(* CODESYS project OSKv1.project

Project tree, tasks and I/O mapping:
  Device : SPK1xx[M01], Production association OWEN, order no. 4, version 3.5.11.54
    application Application
      libraries: Standard, * (System); VisuDialogs, * (System); Standard64, * (System); Util, * (System); VisuKeyboard_En-Ru, 1.3.0.0 (PC Prolog); OwenArchiverErrors, 3.5.4.3 (Production association OWEN); Mx110 Assistant, 3.5.4.12 (Production association OWEN)
      task MainTask (cyclic, interval t#20ms, priority 1) calls PLC_PRG, SteamBlow, DryMode, PaintMode, Utils, PID_controller, AnalogSensHandle, Emrg
      task TrendRecordingTask (cyclic, interval 100 ms, priority 31) calls VisuTrendStorageAccess.GlobalInstances.g_TrendRecordingManager.CyclicCall
      task AlarmManagerTask (cyclic, interval 50 ms, priority 31) calls AlarmManager.Alarm_Prg
      task VISU_TASK (cyclic, interval 100 ms, priority 31) calls VisuElems.Visu_Prg
      task OwenArchiver (cyclic, interval T#100ms, priority 10) calls OwenArchiverDrivers.Archive_Prg
      program PLC_PRG [LD]
      visualisation Humidifier
      program PaintMode [ST]
      global variables GVL
      program DryMode [ST]
      Trend Recording Manager
        Trend_Trend1
      visualisation Chiller
      visualisation StartScreen
      visualisation MainMenu
      program SteamBlow [ST]
      visualisation Trend
      visualisation VENT
      visualisation Settings
      Alarm Configuration
        alarm class Error (priority 10, acknowledge REP_ACK)
        alarm class Warning (priority 30, acknowledge REP)
        alarm class Info (priority 100, acknowledge REP)
        AlarmStorage
        text list Emergencies
        alarm group Emergencies
            0 [Error]: Comparison Equal, ExpressionToCompare TRUE, Expression GVL.InNetEmerg - "Авария по защитам"
            1 [Error]: Comparison Equal, ExpressionToCompare TRUE, Expression Emrg.PhaseEmerg - "Аваря по реле контроля фаз"
            2 [Error]: Comparison Equal, ExpressionToCompare TRUE, Expression Emrg.HeatEmerg - "Нет нагрева"
            3 [Error]: Comparison Equal, ExpressionToCompare TRUE, Expression Emrg.PressureEmerg - "Реле давления"
            4 [Error]: Comparison Equal, ExpressionToCompare TRUE, Expression GVL.TempSensError - "Ошибка датчика температуры"
            5 [Error]: Comparison Equal, ExpressionToCompare TRUE, Expression GVL.HumidSensEmerg - "Ошибка датчика влажности"
            6 [Error]: Comparison Equal, ExpressionToCompare TRUE, Expression GVL.PressBoundsEemrg - "Ошибка давления в камере"
      visualisation DryProgs
      program Utils [ST]
      visualisation DeviceCheck
      visualisation DeviceCheck_2
      program PID_controller [ST]
      visualisation Archive
      program Emrg [ST]
      program AnalogSensHandle [ST]
      visualisation Emergencies
      image pool Images
    OwenRTC : OwenRTC, Production association OWEN, version 3.5.11.5001
        input  Application.PLC_PRG.PLC_DATE : ARRAY [0..80] OF BYTE  // Format Date
        input  Application.PLC_PRG.PLC_TIME : ARRAY [0..80] OF BYTE  // Format Time
        unmapped channels: Year, Month, Day, Hour, Minute, Second, Day of Week, Week of Year, UTC Offset, NTP Enabled, NTP Error, System Timer, New Year, New Month, New Day, New Hour, New Minute, New Second, New UTC Offset, Set Settings DT, Enable NTP, Prefer Server
    OwenCloud : OwenCloud, Production association OWEN, version 3.5.11.5001
        unmapped channels: OwenCloud enabled, Enable OwenCloud, Token
    Buzzer : Buzzer, Production association OWEN, version 3.5.11.5001
        unmapped channels: Buzzer enabled, Enable Buzzer
    Drives : Drives, Production association OWEN, version 3.5.11.5001
        input  Application.PLC_PRG.USBMounted : BIT  // MMC Mounted
        input  Application.PLC_PRG.USBUnmountDone : BIT  // MMC Unmount done
        output Application.Utils.DrivesOn : BIT  // Enable Drives
        output Application.PLC_PRG.USBUnmount : BIT  // MMC Unmount
        unmapped channels: FS size, FS used, FS free, USB Mounted, USB Unmount done, USB size, USB used, USB free, MMC size, MMC used, MMC free, USB Unmount
    Network : Network, Production association OWEN, version 3.5.11.5001
        unmapped channels: DHCP enabled, IP, Mask, Gateway, MAC, Hostname, Enable DHCP, New IP, New Mask, New Gateway, New Hostname, Set Settings
    Screen : Screen, Production association OWEN, version 3.5.11.5001
        unmapped channels: Get Brightness, Dim time, Off time, Full brightness, Dim brightness, Off brightness, Dim visu name, Off visu name, On visu name, Wake up
    Debug : Debug, Production association OWEN, version 3.5.11.5001
        unmapped channels: RAM used, RAM free, Open files, Processor usage, Core temp, Enable Debug, Debug pause
    Info : Info, Production association OWEN, version 3.5.11.5002
        unmapped channels: VENDOR, DEVICE, SERIAL, RUNTIME, FIRMWARE, LINUX, TARGET, PROJECT, AUTHOR, VERSION, PROFILE, LASTCHANGES
    Watchdog : Watchdog, Production association OWEN, version 3.5.11.5001
        unmapped channels: Exception Handling, Last Exception Code, Last Exception Description, Last Exception Time, Hardware Watchdog Flag, Reboot
    OwenArchiver : OwenArchiver, Production association OWEN, version 3.5.4.9
        output Application.PLC_PRG.StartArchive : BIT  // Запустить архиватор
        unmapped channels: Команда записи, Запись лога отладки, Путь архивации, Имя архива, Код последней ошибки, Архиватор работает, Использование буфера записи, Размер архива
      CSVFormat : CSVFormat, Production association OWEN, version 3.5.4.9
      REAL_Variable : REAL Variable, Production association OWEN, version 3.5.4.9
          settings: Описание переменной = 'Temperatura v kamere'
          output Application.GVL.ChamberFinalTemp : REAL  // Переменная
      REAL_Variable_1 : REAL Variable, Production association OWEN, version 3.5.4.9
          settings: Описание переменной = 'Vlazhnost'
          output Application.GVL.InAHumInside : REAL  // Переменная
      INT_Variable : INT Variable, Production association OWEN, version 3.5.4.9
          settings: Описание переменной = 'Rezhim raboti'
          output Application.GVL.Mode : INT  // Переменная
      NetEmegAch : BYTE Variable, Production association OWEN, version 3.5.4.9
          settings: Описание переменной = 'Avaria po zachitam'
          output Application.Emrg.NetEmergByte : BYTE  // Переменная
      PhaseEmergArch : BYTE Variable, Production association OWEN, version 3.5.4.9
          settings: Описание переменной = 'Rele cntrolya faz'
          output Application.Emrg.PhaseEmergByte : BYTE  // Переменная
      ChillerEmergArc : BYTE Variable, Production association OWEN, version 3.5.4.9
          settings: Описание переменной = 'Avariya chillera'
          output Application.GVL.InChillerEmerByte : BYTE  // Переменная
      HumidEmergArch : BYTE Variable, Production association OWEN, version 3.5.4.9
          settings: Описание переменной = 'Avariya uvlazhnitelya'
          output Application.GVL.InHumidEmergByte : BYTE  // Переменная
      PressureEmergArch : BYTE Variable, Production association OWEN, version 3.5.4.9
          settings: Описание переменной = 'Rele davleniya'
          output Application.Emrg.PressureEmergByte : BYTE  // Переменная
      UpperFilterArch : BYTE Variable, Production association OWEN, version 3.5.4.9
          settings: Описание переменной = 'Zagrayznenie verhnego filtra'
          output Application.Emrg.UpperFilterOutByte : BYTE  // Переменная
      LowerFilterArch : BYTE Variable, Production association OWEN, version 3.5.4.9
          settings: Описание переменной = 'Zagryaznenie nizhnego filtra'
          output Application.Emrg.LowerFilterOutByte : BYTE  // Переменная
      TempSensErrorArch : BYTE Variable, Production association OWEN, version 3.5.4.9
          settings: Описание переменной = 'Oshibka datchika temperaturi'
          output Application.GVL.TempSensErrorByte : BYTE  // Переменная
      HumidSensEmergArch : BYTE Variable, Production association OWEN, version 3.5.4.9
          settings: Описание переменной = 'Oshibka datchika vlazhnosti'
          output Application.GVL.HumidSensEmergByte : BYTE  // Переменная
      HeatEmergArch : BYTE Variable, Production association OWEN, version 3.5.4.9
          settings: Описание переменной = 'Net nagreva'
          output Application.Emrg.HeatEmergByte : BYTE  // Переменная
      PressureBoundsEmergArch : BYTE Variable, Production association OWEN, version 3.5.4.9
          settings: Описание переменной = 'Davlenie vishlo za ramki'
          output Application.GVL.PressBoundsEemrgByte : BYTE  // Переменная
    Modbus_COM : Modbus COM, 3S - Smart Software Solutions GmbH, version 3.5.11.20
        settings: DataBits = 8; StopBits = 1; ComPort = 1
      Modbus_Master_COM_Port : Modbus Master, COM Port, 3S - Smart Software Solutions GmbH, version 3.5.11.20
          settings: Transmission = 'RTU'; ResponseTimeout = 1000; TimeBetweenFrames = 10; Auto-restart communication = TRUE
        MV110_8A : MV110-8A, Production association OWEN, version 3.5.11.04
            input  Application.GVL.InAChamberTemp : REAL  // Измеренное значение
            input  Application.GVL.InAHExchanger : REAL  // Измеренное значение
            input  Application.GVL.InAEntryTemp : REAL  // Измеренное значение
            input  Application.GVL.InAHumInside : REAL  // Измеренное значение
            input  Application.GVL.InAChambPressure : REAL  // Измеренное значение
            input  Application.GVL.InAHumOutside : REAL  // Измеренное значение
            input  Application.GVL.InAFBHeatGate : REAL  // Измеренное значение
            input  Application.GVL.inAFBCoolGate : REAL  // Измеренное значение
            unmapped channels: Channels1_3State, Channels4_6State, Channels7_8State, Отключить модуль, Флаг ошибки, Код статуса, Код статуса, Код статуса, Код статуса, Код статуса, Код статуса, Код статуса, Код статуса, Циклическое время, Циклическое время, Циклическое время, Циклическое время, Циклическое время, Циклическое время, Циклическое время, Циклическое время
        MU110_16R_K : MU110-16R_K, Production association OWEN, version 3.5.11.04
            settings: SlaveAddress = 17; ResponseTimeout = 1000; UseExtendedFunctionCodes = TRUE
            output Application.GVL.OutInflowFan : BOOL  // Маска выходов (запись).Выход 1
            output Application.GVL.OutExhaustFan : BOOL  // Маска выходов (запись).Выход 2
            output Application.GVL.OutLight1 : BOOL  // Маска выходов (запись).Выход 3
            output Application.GVL.OutLight2 : BOOL  // Маска выходов (запись).Выход 4
            output Application.GVL.OutChiller : BOOL  // Маска выходов (запись).Выход 5
            output Application.GVL.OutHumid : BOOL  // Маска выходов (запись).Выход 6
            output Application.GVL.OutEmergLamp : BOOL  // Маска выходов (запись).Выход 7
            output Application.GVL.OutAirPump : BOOL  // Маска выходов (запись).Выход 8
            output Application.GVL.OutModeGate : BOOL  // Маска выходов (запись).Выход 9
            output Application.GVL.OutHeatGate : BOOL  // Маска выходов (запись).Выход 10
            output Application.GVL.OutCoolGate : BOOL  // Маска выходов (запись).Выход 11
            unmapped channels: rMask, wMask, wAlarmState, wAlarmState, Отключить модуль, Флаг ошибки, Маска выходов (запись), Маска выходов (чтение), Аварийное состояние выходов, Запись аварийного состояния
        MV110_16D_DN : MV110-16D_DN, Production association OWEN, version 3.5.11.04
            settings: SlaveAddress = 18; ResponseTimeout = 1000; UseExtendedFunctionCodes = TRUE
            input  Application.GVL.InChillerPwr : BOOL  // Маска входов.Вход 1
            input  Application.GVL.InChillerPump : BOOL  // Маска входов.Вход 2
            input  Application.GVL.InChillerCompressor : BOOL  // Маска входов.Вход 3
            input  Application.GVL.InChillerEmer : BOOL  // Маска входов.Вход 4
            input  Application.GVL.InHumidPwr : BOOL  // Маска входов.Вход 5
            input  Application.GVL.InHumidEmerg : BOOL  // Маска входов.Вход 6
            input  Application.GVL.InFireSteam : BOOL  // Маска входов.Вход 7
            input  Application.GVL.InModeGatePaint : BOOL  // Маска входов.Вход 9
            input  Application.GVL.InModeGateDry : BOOL  // Маска входов.Вход 10
            input  Application.GVL.InPhaseControl : BOOL  // Маска входов.Вход 11
            input  Application.GVL.InNetEmerg : BOOL  // Маска входов.Вход 12
            input  Application.GVL.InChamberPressure : BOOL  // Маска входов.Вход 13
            input  Application.GVL.InUpperFilter : BOOL  // Маска входов.Вход 14
            input  Application.GVL.InLowerFilter : BOOL  // Маска входов.Вход 15
            unmapped channels: Mask, rCounters, wCounter1, wCounter1, wCounter2, wCounter2, wCounter3, wCounter3, wCounter4, wCounter4, wCounter5, wCounter5, wCounter6, wCounter6, wCounter7, wCounter7, wCounter8, wCounter8, wCounter9, wCounter9, wCounter10, wCounter10, wCounter11, wCounter11, wCounter12, wCounter12, wCounter13, wCounter13, wCounter14, wCounter14, wCounter15, wCounter15, wCounter16, wCounter16, Отключить модуль, Флаг ошибки, Маска входов, Значение счетчика, Запись значения счетчика, Команда на запись,
              Значение счетчика, Запись значения счетчика, Команда на запись, Значение счетчика, Запись значения счетчика, Команда на запись, Значение счетчика, Запись значения счетчика, Команда на запись, Значение счетчика, Запись значения счетчика, Команда на запись, Значение счетчика, Запись значения счетчика, Команда на запись, Значение счетчика, Запись значения счетчика, Команда на запись, Значение счетчика, Запись значения счетчика, Команда на запись, Значение счетчика, Запись значения счетчика, Команда на запись, Значение счетчика, Запись значения счетчика, Команда на запись, Значение счетчика, Запись значения счетчика, Команда на запись, Значение счетчика, Запись значения счетчика, Команда на запись, Значение счетчика, Запись значения счетчика, Команда на запись, Значение счетчика, Запись значения счетчика, Команда на запись, Значение счетчика,
              Запись значения счетчика, Команда на запись, Значение счетчика, Запись значения счетчика, Команда на запись
  text list GlobalTextList
  image pool ImagePool
  5ce3da45-db07-42e7-a21c-a00fff4ed8f6|Gear.png
  5ce3da45-db07-42e7-a21c-a00fff4ed8f6|G:\2019.png
  5ce3da45-db07-42e7-a21c-a00fff4ed8f6|G:\123.png
  5ce3da45-db07-42e7-a21c-a00fff4ed8f6|G:\36185-200.png
  5ce3da45-db07-42e7-a21c-a00fff4ed8f6|123.png
  5ce3da45-db07-42e7-a21c-a00fff4ed8f6|2019.png
  5ce3da45-db07-42e7-a21c-a00fff4ed8f6|36185-200.png
*)

// Device/Application/GVL
{attribute 'qualified_only'}
VAR_GLOBAL
	Mode : INT; // 0 = останов 1 = окраска 2 = сушка 3 = продув по парам 4 = авария
	
	PIDTargetTemp : REAL;
	PIDEnable : BOOL;
	ChamberFinalTemp : REAL;
	HExchangerFinalTemp : REAL;
	EntryFinalTemp : REAL;
	
	HeatBlock : BOOL;
	Emergency : BOOL;
	NotEmerg : bool;
	ExhFanD : INT;
	TempSensError : BOOL;
	TempSensErrorByte : BYTE;
	PressBoundsEemrg : BOOL;
	PressBoundsEemrgByte : BYTE;
	HumidSensEmerg : BOOL;
	HumidSensEmergByte : BYTE;
	
	OutInflowFan : BOOL;
	OutExhaustFan : BOOL;
	OutLight1 : BOOL;
	OutLight2 : BOOL;
	OutChiller : BOOL;
	OutHumid : BOOL;
	OutEmergLamp : BOOL;
	OutModeGate : BOOL;
	OutAirPump : BOOL;
	OutHeatGate : BOOL;
	OutCoolGate : BOOL;
	
	InChillerPwr : BOOL;
	InChillerPump : BOOL;
	InChillerCompressor : BOOL;
	InChillerEmer : BOOL;
	InChillerEmerByte : BYTE;
	
	InHumidPwr : BOOL;
	InHumidEmerg : BOOL;
	InHumidEmergByte : BYTE;
	InFireSteam : BOOL;
	InModeGatePaint : BOOL;
	InModeGateDry : BOOL;
	InPhaseControl : BOOL;
	InNetEmerg : BOOL;
	InChamberPressure : BOOL;
	InUpperFilter : BOOL;
	InLowerFilter : BOOL;
	
	
	InAChamberTemp : REAL;
	InAHExchanger : REAL;
	InAEntryTemp : REAL;
	InAFBHeatGate : REAL;
	inAFBCoolGate : REAL;
	InAHumOutside : REAL;
	InAHumInside : REAL;
	InAChambPressure : REAL;
	
END_VAR

// Device/Application/PLC_PRG
PROGRAM PLC_PRG
VAR
	PLC_DATE : STRING(80);
	PLC_TIME : STRING(80);
	dwLightColorToggle : DWORD := 16#FFFFFF00;
	dwOffColorToggle : DWORD := 16#FFFFFFFF;
	ColorGreen : dword := 16#FF009900;
	xButtonLight1 : BOOL;
	xButtonLight2 : BOOL;
	
	StartArchive : BOOL;
	USBMounted: BOOL;
	USBUnmount : BOOL;
	USBUnmountDone : BOOL;
END_VAR
VAR RETAIN
	Light1Ret: BOOL;
	Light2Ret: BOOL;
END_VAR

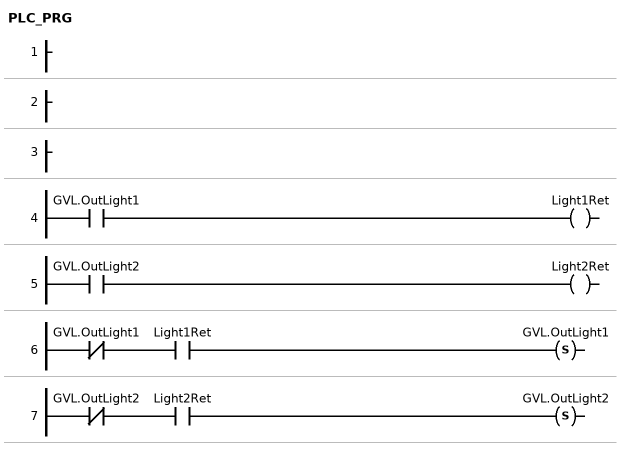
// NETWORK 1

// NETWORK 2

// NETWORK 3

// NETWORK 4
Light1Ret := GVL.OutLight1;

// NETWORK 5
Light2Ret := GVL.OutLight2;

// NETWORK 6
GVL.OutLight1 S= NOT GVL.OutLight1 AND Light1Ret;

// NETWORK 7
GVL.OutLight2 S= NOT GVL.OutLight2 AND Light2Ret;

END_PROGRAM

// Device/Application/SteamBlow
PROGRAM SteamBlow
VAR
	Stage: INT;
	FanCD : TON;
	FanCDStart : BOOL;
	FanCDOut : BOOL;
	
END_VAR

IF .GVL.InFireSteam THEN
	.GVL.Mode := 3;
	Stage := 1;
END_IF

IF (.GVL.InModeGateDry AND Stage = 1) THEN .GVL.OutModeGate := TRUE; END_IF;

IF (.GVL.InModeGatePaint AND Stage = 1) THEN
	.GVL.OutInflowFan := TRUE;
	FanCDStart := TRUE;
	Stage := 2;
END_IF;

FanCD(IN := FanCDStart, PT:= INT_TO_TIME(.GVL.ExhFanD*1000),Q => FanCDOut);

IF FanCDOut THEN
	.GVL.OutExhaustFan := true;
	FanCDStart := FALSE;
END_IF

IF NOT .GVL.InFireSteam AND Stage <> 0 THEN
	.GVL.OutExhaustFan := FALSE;
	.GVL.OutInflowFan := FALSE;
	FanCDStart := FALSE;
	Stage := 0;
	.GVL.Mode := 0;
END_IF

END_PROGRAM

// Device/Application/DryMode
PROGRAM DryMode
VAR
	Modes : ARRAY [0..3] OF WSTRING := ["Пусто","Окраска","Сушка","Продув"];	

	ChosenProg : WORD;
	DryModeM : BOOL;	
	
	NewName : WSTRING;
	SaveName : BOOL;
	ProgChanged : BOOL;	
	SelectedProg: WORD;
	ProgSave : BOOL;
	CurrentName : WSTRING;
	StepTimeLeft : TIME;
	CurStepTime: TIME;
	
	Buffer : ARRAY [1..3,1..10] OF REAL;
	ChooseProg : BOOL;
	
	index: WORD;
	Stage : WORD;
	
	DryTimer : TON;
	DryTimerM : BOOL;
	DryTimerOut : BOOL;
	TempCmp : BOOL;
	
	i: WORD;
	j: WORD;
END_VAR
VAR RETAIN
		// 1 - параметр, 2 - шаг, 3 - программа
	DryPrograms : ARRAY [1..3,1..10,1..10] OF REAL;
	Progs : ARRAY [0..10] OF WSTRING:= ["Выберите программу"];
END_VAR

CurrentName:= Progs[ChosenProg];

IF (ProgChanged = TRUE AND SelectedProg <> 0) THEN
	FOR i:=1 TO 3 BY 1 DO
		FOR j:=1 TO 10 BY 1 DO
			Buffer[i,j] := DryPrograms[i,j,SelectedProg];
		END_FOR;
	END_FOR;
	ProgChanged := FALSE;
END_IF

IF (ProgSave = TRUE AND SelectedProg <> 0) THEN
	FOR i:=1 TO 3 BY 1 DO
		FOR j:=1 TO 10 BY 1 DO
			DryPrograms[i,j,SelectedProg] := Buffer[i,j];
		END_FOR;
	END_FOR;
	ProgSave := FALSE;
END_IF

IF (SaveName = TRUE AND SelectedProg <> 0) THEN
	Progs[SelectedProg] := NewName;
	SaveName := FALSE;
END_IF

IF (ChooseProg = TRUE) THEN
	ChosenProg := SelectedProg;
	ChooseProg := FALSE;
END_IF


IF (Stage = 0 AND .GVL.Mode = 2) THEN index := 1; Stage := 2; DryModeM := TRUE; END_IF; //1

//Если след режим = окр или продув, заслонка = сушка, то выкл вент и заслонку в окраску  2
IF (.GVL.InModeGateDry AND (DryPrograms[1,index,ChosenProg] = 1 OR DryPrograms[1,index,ChosenProg] = 3) AND Stage = 2) THEN 
	.GVL.OutModeGate := TRUE;
	.GVL.OutInflowFan := FALSE;
	.GVL.OutExhaustFan := FALSE;
END_IF;

//Если некст режим = сушка, заслонка = окраска, то выкл вент и заслонку в сушку  3
IF (.GVL.InModeGatePaint AND DryPrograms[1,index,ChosenProg] = 2 AND Stage = 2) THEN 
	.GVL.OutModeGate := FALSE;
	.GVL.OutInflowFan := FALSE;
	.GVL.OutExhaustFan := FALSE;
END_IF;

//Если А[1][index][ChosenProg] = 2 и правильно стоит режимная  4
IF (.GVL.InModeGateDry AND DryPrograms[1,index,ChosenProg] = 2 AND Stage = 2 ) THEN
	IF index > 1 THEN
		IF DryPrograms[2,index,ChosenProg] < DryPrograms[2,index,ChosenProg-1] THEN
			TempCmp := TRUE;
		ELSE TempCmp := FALSE;
		END_IF
	END_IF
	.GVL.PIDTargetTemp := DryPrograms[2,index,ChosenProg];
	.GVL.PIDEnable := TRUE;
	
	.GVL.OutInflowFan := TRUE;
	Stage:=4;
END_IF

// если некст режим = 1 или 3  и правильно стоит режимная  5
IF (.GVL.InModeGatePaint AND (DryPrograms[1,index,ChosenProg] = 1 OR DryPrograms[1,index,ChosenProg] = 3) AND Stage = 2 ) THEN 
	IF index > 1 THEN
		IF DryPrograms[2,index,ChosenProg] < DryPrograms[2,index,ChosenProg-1] THEN
			TempCmp := TRUE;
		ELSE TempCmp := FALSE;
		END_IF
	END_IF
	
	.GVL.OutInflowFan := TRUE;
	.GVL.OutExhaustFan := TRUE;
	DryTimerM := TRUE; //Если режим "вытяжка - вкл", то таймер запускается сразу после начала пункта меню (не дожидаясь достижения температуры).
	Stage := 4;
	.GVL.PIDTargetTemp := DryPrograms[2,index,ChosenProg];
	.GVL.PIDEnable := TRUE;
END_IF;


//если режим - сушка и достигли темп  6
IF (Stage = 4 AND DryPrograms[1,index,ChosenProg] = 2 AND ((.GVL.ChamberFinalTemp < DryPrograms[2,index,ChosenProg] AND TempCmp) OR (.GVL.ChamberFinalTemp > DryPrograms[2,index,ChosenProg] AND NOT TempCmp)) ) THEN
	DryTimerM := TRUE;
END_IF

//В режиме продув остановка по дост темп  7
IF (Stage = 4 AND DryPrograms[1,index,ChosenProg] = 3 AND ((.GVL.ChamberFinalTemp < DryPrograms[2,index,ChosenProg] AND TempCmp) OR (.GVL.ChamberFinalTemp > DryPrograms[2,index,ChosenProg] AND NOT TempCmp))) THEN
	DryTimerM := FALSE;
	Stage := 0;	
	.GVL.OutHeatGate := FALSE;
	.GVL.OutCoolGate := FALSE;
	.GVL.OutInflowFan := FALSE;
	.GVL.OutExhaustFan := FALSE;
	.GVL.Mode := 0;
	DryModeM := FALSE;
	index := 0;
	.GVL.PIDEnable := FALSE;
END_IF

StepTimeLeft := REAL_TO_TIME(DryPrograms[3,index,ChosenProg]*1000) - CurStepTime;

DryTimer(IN := DryTimerM, PT:= REAL_TO_TIME(DryPrograms[3,index,ChosenProg]*1000),ET => CurStepTime,Q => DryTimerOut);

// переход к след шагу по таймеру при режимах 1 и 2   8
IF (DryTimerOut AND DryPrograms[1,index,ChosenProg] <> 3) THEN
	DryTimerM := FALSE;
	Stage := 2;
	index:= index + 1;
END_IF

//если таймер достиг и режим продув то законч работу  9
IF (DryTimerOut AND DryPrograms[1,index,ChosenProg] = 3) THEN
	DryTimerM := FALSE;
	Stage := 0;
	.GVL.OutHeatGate := FALSE;
	.GVL.OutCoolGate := FALSE;
	.GVL.OutInflowFan := FALSE;
	.GVL.OutExhaustFan := FALSE;
	.GVL.Mode := 0;
	DryModeM := FALSE;
	index := 0;
	.GVL.PIDEnable := FALSE;
END_IF

//Handle stop button
IF (.GVL.Mode <> 2 AND stage <> 0) THEN
stage := 0;
.GVL.OutHeatGate := FALSE;
.GVL.OutCoolGate := FALSE;
.GVL.OutExhaustFan := FALSE;
.GVL.OutInflowFan := FALSE;
DryTimerM := FALSE;
DryModeM := FALSE;
index := 0;
.GVL.PIDEnable := FALSE;
END_IF

END_PROGRAM

// Device/Application/PaintMode
PROGRAM PaintMode
VAR
	ExhFanT : TON;
	ExhFanM : BOOL;
	
	ExhFanOut : BOOL;
	
	PaintModeM : BOOL;
	
	ChillT : TON;
	ChillM : BOOL;
	ChillOut : BOOL;
	ChillOK :BOOL;
	ChillHigh : REAL;
	ChillLow : REAL;
	
	Stage : int := 0;
	trig : R_TRIG;

	HumidMax : REAL;
	HumidOk : bool;
	
	TempInc :BOOL;
	TempDec :BOOL;
	TempIncS : BOOL;
	TempDecS : BOOL;
END_VAR
VAR RETAIN
	HumidTarget : INT;
	HumidDiff : INT;
	
	PaintPIDTarget : REAL;
	
	ChillHDiff : REAL;
	ChillLDiff : REAL;
	ChillCD : DINT;
END_VAR

// После нажатия кнопки, проверяется положение режимной заслонки и, при необходимости, она переводится в положение "Окраска".
IF (Stage = 0 AND .GVL.Mode = 1) THEN stage:= 1; PaintModeM := true; END_IF;


IF (.GVL.InModeGateDry AND Stage = 1 AND .GVL.Mode = 1) THEN .GVL.OutModeGate := TRUE; END_IF;

// По окончании перевода, запускается приточный вентилятор и, 
IF (.GVL.InModeGatePaint AND Stage = 1 AND .GVL.HeatBlock = FALSE) THEN 
	Stage := 2;
	.GVL.OutExhaustFan := TRUE;
	ExhFanM:= TRUE;
END_IF;

//через несколько секунд, запускается вытяжной вентилятор и клапан подачи воздуха. 
ExhFanT(IN := ExhFanM, PT:= INT_TO_TIME(.GVL.ExhFanD*1000),Q => ExhFanOut);
IF (ExhFanOut = TRUE AND Stage = 2) THEN 
	.GVL.OutInflowFan := TRUE;
	.GVL.OutAirPump := TRUE;
	Stage := 3;
	ExhFanM:= FALSE;
	.GVL.PIDTargetTemp := PaintPIDTarget;
	.GVL.PIDEnable := TRUE;
END_IF;

//настройка температуры кнопками с панели
IF (TempInc = TRUE)THEN
	PaintPIDTarget := PaintPIDTarget + 1;
	TempInc := FALSE;
END_IF
IF (TempDec = TRUE)THEN
	PaintPIDTarget := PaintPIDTarget - 1;
	TempDec := FALSE;
END_IF
IF (TempIncS = TRUE)THEN
	PaintPIDTarget := PaintPIDTarget + 0.1;
	TempIncS := FALSE;
END_IF
IF (TempDecS = TRUE)THEN
	PaintPIDTarget := PaintPIDTarget - 0.1;
	TempDecS := FALSE;
END_IF

HumidMax := HumidTarget + HumidDiff;

ChillHigh := PaintPIDTarget + ChillHDiff;
ChillLow := PaintPIDTarget + ChillLDiff;

IF (.GVL.InHumidEmerg OR NOT .GVL.InHumidPwr OR .GVL.HumidSensEmerg) THEN
	HumidOk := FALSE;
	.GVL.OutHumid := FALSE;
ELSE HumidOk := TRUE;
END_IF

IF (.GVL.InChillerEmer OR NOT .GVL.InChillerPwr) THEN
	ChillOK := FALSE;
	.GVL.OutChiller := FALSE;
ELSE ChillOK:= TRUE;
END_IF

// В случае, если заслонка находится в положении "0% нагрев", а температура окраски выше заданной более чем на ХХ градуса, включается чиллер
IF (.GVL.InAFBHeatGate < 5 AND stage = 3 AND .GVL.ChamberFinalTemp > ChillHigh AND ChillOK = TRUE) THEN
		.GVL.OutChiller := TRUE;
		Stage := 4;
		.GVL.HeatBlock := TRUE;
END_IF

// И продолжает работать, пока температура не упадет на ХХ градуса ниже температуры ставки. Затем чиллер выключается и запускается внутренний таймер на УУ минут
IF (.GVL.ChamberFinalTemp < ChillLow AND stage = 4) THEN
		.GVL.OutChiller := FALSE;
		ChillM := TRUE;
		stage := 5;
END_IF
ChillT(IN := ChillM, PT:= DINT_TO_TIME(ChillCD*60000),Q => ChillOut);

// По окончании работы этого таймера допускается нагрев воздуха посредством теплообменника
IF (ChillOut = TRUE) THEN
		ChillM := FALSE;
		stage := 0;
		.GVL.HeatBlock := FALSE;
END_IF

// Поддержка влажности
IF (.GVL.InAHumInside > HumidMax AND stage = 3) THEN
		.GVL.OutHumid := FALSE;
END_IF

IF (.GVL.InAHumInside < HumidTarget AND stage = 3 AND HumidOk = TRUE) THEN
		.GVL.OutHumid := TRUE;
END_IF

//Handle stop button
IF (.GVL.Mode <> 1 AND stage <> 0) THEN
stage := 0;
.GVL.OutHeatGate := FALSE;
.GVL.OutCoolGate := FALSE;
.GVL.OutExhaustFan := FALSE;
.GVL.OutInflowFan := FALSE;
.GVL.OutAirPump := FALSE;
.GVL.OutChiller := FALSE;
.GVL.OutHumid := FALSE;
ChillM := FALSE;
ExhFanM := FALSE;
PaintModeM := FALSE;
.GVL.PIDEnable := FALSE;
END_IF

END_PROGRAM

// Device/Application/Utils
PROGRAM Utils
VAR
	GateMode : WSTRING;
	PressureTMR : TON;
	PressureM : BOOL;
	PressureOutM : BOOL;
	
	DrivesOn: BOOL;
	timeR : UINT;
	
	PressureHigh : WORD;
	PressureLow: WORD;
	
	ManualBlock : BOOL;
	
	ColorYelllow : DWORD := 16#FFFFFF00;
	ColorWhite : DWORD := 16#FFFFFFFF;
	ColorGreen : DWORD := 16#FF009900;
	ColorRed : DWORD := 16#FFFF3300;
	
	CurrentChillerColor : DWORD;
	CurrentHumidColor: DWORD;
	CurrentVentColor: DWORD;
	
	ModeGateImg : BOOL;
	NotInflowFan : BOOL;
	NotExhaustFan : BOOL;
END_VAR

IF .GVL.InModeGateDry THEN
	ModeGateImg := FALSE;
ELSIF .GVL.InModeGatePaint THEN
	ModeGateImg := TRUE;
END_IF;

DrivesOn:=true;

NotInflowFan := NOT .GVL.OutInflowFan;
NotExhaustFan := NOT .GVL.OutExhaustFan;

IF .GVL.InChillerEmer THEN
	CurrentChillerColor := ColorRed;
ELSIF .GVL.OutChiller THEN
	CurrentChillerColor := ColorGreen;
ELSE
	CurrentChillerColor := ColorWhite;
END_IF;

IF .GVL.InHumidEmerg THEN
	CurrentHumidColor := ColorRed;
ELSIF .GVL.OutHumid THEN
	CurrentHumidColor := ColorGreen;
ELSE
	CurrentHumidColor := ColorWhite;
END_IF;

IF .GVL.Mode > 2 THEN
	CurrentVentColor := ColorRed;
ELSIF .GVL.Mode > 0 THEN
	CurrentVentColor := ColorGreen;
ELSE
	CurrentVentColor := ColorWhite;
END_IF;

IF .GVL.InModeGateDry THEN
GateMode := "Сушка";
ELSIF .GVL.InModeGatePaint THEN
        GateMode := "Окраска";
ELSE
        GateMode := "Переход";
END_IF;


IF (.GVL.OutInflowFan OR .GVL.OutExhaustFan) AND (.GVL.InAChambPressure > PressureHigh OR .GVL.InAChambPressure < PressureLow) THEN
	PressureM := TRUE;
ELSE
	PressureM := FALSE;
END_IF;

PressureTMR(IN := PressureM, PT:= INT_TO_TIME(20000),Q => PressureOutM);

IF PressureOutM THEN
	.GVL.PressBoundsEemrg := TRUE;
ELSE .GVL.PressBoundsEemrg := FALSE;
END_IF

IF .GVL.Mode <> 0 THEN
	ManualBlock := TRUE;
ELSE ManualBlock := FALSE;
END_IF

END_PROGRAM

// Device/Application/PID_controller
PROGRAM PID_controller
VAR
	PeriodicTMR : TON;
	TMRIn : BOOL;
	TMROut : BOOL;
	TMRCurr : TIME;

	Delta : REAL;
	PIDArray : ARRAY [1..11] OF REAL;
	ArraySum : REAL;
	
	PropComponent : REAL;
	IntComponent : REAL;
	FinalEqus : REAL;
	FinalResult : REAL;
	
	i : INT;
END_VAR
VAR RETAIN
	KI : WORD;
	KP : WORD;
	Tau : WORD;
END_VAR

PeriodicTMR(IN := TMRIn, PT:= WORD_TO_TIME(Tau*1000),ET => TMRCurr,Q => TMROut);
IF TMRIn =  FALSE AND .GVL.PIDEnable = TRUE THEN
	TMRIn := TRUE;
END_IF
IF .GVL.PIDEnable = FALSE THEN
	FOR i:=1 TO 10 BY 1 DO
		PIDArray[i] := 0;
	END_FOR;
END_IF
IF TMROut THEN
	ArraySum := 0;
	Delta := .GVL.ChamberFinalTemp - .GVL.PIDTargetTemp;
	PIDArray[11] := Delta;
	FOR i:=1 TO 10 BY 1 DO
		PIDArray[i] := PIDArray[i+1];
		ArraySum:=ArraySum+PIDArray[i];
	END_FOR;
	
	PropComponent := Delta * KP;
	IntComponent := ArraySum * KI;
	
	FinalEqus := (PropComponent + IntComponent) / 100;
	
	IF FinalEqus > 100 THEN
		FinalResult := 100;
	ELSIF FinalEqus < -100 THEN
		FinalResult := -100;
		ELSE FinalResult := FinalEqus;
	END_IF
	TMRIn := FALSE;
END_IF

IF .GVL.PIDEnable THEN
	IF FinalResult < 0 THEN
		IF .GVL.inAFBHeatGate <> FinalResult THEN
			.GVL.OutHeatGate := TRUE;
		ELSE .GVL.OutHeatGate := FALSE;
		END_IF
	ELSIF .GVL.inAFBCoolGate <> FinalResult THEN
		.GVL.OutCoolGate := TRUE;
		.GVL.OutHeatGate := TRUE;
		ELSE .GVL.OutCoolGate := FALSE;
			.GVL.OutHeatGate := FALSE;
	END_IF
END_IF

END_PROGRAM

// Device/Application/AnalogSensHandle
PROGRAM AnalogSensHandle
VAR
END_VAR

IF .GVL.TempSensError THEN
	.GVL.ChamberFinalTemp := .GVL.InAEntryTemp / 10;
ELSE .GVL.ChamberFinalTemp := .GVL.InAChamberTemp / 10;
END_IF

GVL.EntryFinalTemp := .GVL.InAEntryTemp /10;
GVL.HExchangerFinalTemp := GVL.InAHExchanger /10;

END_PROGRAM

// Device/Application/Emrg
PROGRAM Emrg
VAR
	PressureEmerg : BOOL; // авария по давлению 4
	PressureEmergByte : BYTE;
	NetEmerg : BOOL ; // авария по реле контроля фаз 1 
	NetEmergByte : BYTE;
	HeatEmerg : BOOL; 
	HeatEmergByte : BYTE;
	PhaseEmerg : BOOL;
	PhaseEmergByte : BYTE;
	                    
	
	PressEmergInv : BOOL;
	PressEmergTON : TON;
	PressEmergStart: BOOL;
	PressEmergOut : BOOL;
	
	PressRelEmergInv : BOOL;
	PressRelEmergTON : TON;
	PressRelEmergStart: BOOL;
	PressRelEmergOut : BOOL;
	
	UpperFilter : TON;
	UpperFilterStart: BOOL;
	UpperFilterOut : BOOL;
	UpperFilterOutByte : BYTE;
	
	LowerFilter : TON;
	LowerFilterStart: BOOL;
	LowerFilterOut : BOOL;
	LowerFilterOutByte : BYTE;
	
	UpperFilterInv : BOOL;
	LowerFilterInv : BOOL;
	
	AcknSelected : BOOL;
	AcknVisible : BOOL;
	EmergHistory : BOOL;
	EmergFixedPos : BOOL;
	
	
END_VAR

PressEmergInv := NOT .GVL.InChamberPressure;
UpperFilterInv := NOT .GVL.InUpperFilter;
LowerFilterInv := NOT .GVL.InLowerFilter;
.GVL.NotEmerg := NOT .GVL.Emergency;

PressureEmergByte := BOOL_TO_BYTE(PressureEmerg);
NetEmergByte:= BOOL_TO_BYTE(NetEmerg);
HeatEmergByte:= BOOL_TO_BYTE(HeatEmerg);
PhaseEmergByte:= BOOL_TO_BYTE(PhaseEmerg);
UpperFilterOutByte := BOOL_TO_BYTE(UpperFilterOut);
LowerFilterOutByte := BOOL_TO_BYTE(LowerFilterOut);
.GVL.TempSensErrorByte := BOOL_TO_BYTE(.GVL.TempSensError);
.GVL.PressBoundsEemrgByte := BOOL_TO_BYTE(.GVL.PressBoundsEemrg);
.GVL.HumidSensEmergByte := BOOL_TO_BYTE(.GVL.HumidSensEmerg);
.GVL.InChillerEmerByte := BOOL_TO_BYTE(.GVL.InChillerEmer);
.GVL.InHumidEmergByte := BOOL_TO_BYTE(.GVL.InHumidEmerg);

//Светофор
.GVL.OutEmergLamp := .GVL.Emergency;
//Общий стоп и запрет
IF .GVL.Emergency THEN
	.GVL.Mode := 4;
END_IF

// Авария по защитам, останов
IF .GVL.InNetEmerg THEN
	NetEmerg := TRUE;
	.GVL.Emergency := TRUE;
ELSE NetEmerg := FALSE;
END_IF

IF .GVL.InPhaseControl THEN
	PhaseEmerg := TRUE;
	.GVL.Emergency := TRUE;
ELSE PhaseEmerg := FALSE;
END_IF

//Авария датчика температуры
IF .GVL.InAChamberTemp > 2000 OR .GVL.InAChamberTemp < -500 THEN
	.GVL.TempSensError := TRUE;
ELSE .GVL.TempSensError := FALSE;
END_IF

//Авария датчика влажности
IF .GVL.InAHumInside > 1000 OR .GVL.InAHumInside < 0 THEN
	.GVL.HumidSensEmerg := TRUE;
	.GVL.Emergency := TRUE;
ELSE .GVL.HumidSensEmerg := FALSE;
END_IF

//Нет нагрева
IF .GVL.InAHExchanger < 200 THEN
	HeatEmerg := TRUE;
	.GVL.Emergency := TRUE;
ELSE HeatEmerg := FALSE;
END_IF

// Задержка срабатывания аварии давления
PressEmergTON(IN := PressEmergStart, PT := INT_TO_TIME(10000), Q=> PressEmergOut);
IF .GVL.OutInflowFan OR .GVL.OutExhaustFan THEN
	PressEmergStart := TRUE;
END_IF
IF PressEmergOut THEN
	PressEmergStart := FALSE;
END_IF

// Авария давления, останов
IF NOT PressEmergStart AND PressEmergInv THEN
	PressureEmerg := TRUE;;
	.GVL.Emergency := TRUE;
ELSE PressureEmerg := FALSE;
END_IF

//Грязный фильтр, индикация 
IF LowerFilterInv THEN
	LowerFilterStart := TRUE;
ELSE LowerFilterStart := FALSE;
END_IF
// грязынй фильтр индикация
IF UpperFilterInv THEN
	UpperFilterStart := TRUE;
ELSE UpperFilterStart := FALSE;
END_IF
LowerFilter(IN := LowerFilterStart, PT := INT_TO_TIME(10000), Q=> LowerFilterOut); // авария грязный фильтр 6
UpperFilter(IN := UpperFilterStart, PT := INT_TO_TIME(10000), Q=> UpperFilterOut); // авария грязный фильтр 5

//сброс глобальной ошибки при отсутствии ош
IF NOT PressureEmerg AND NOT NetEmerg AND NOT PhaseEmerg AND NOT .GVL.InNetEmerg AND NOT .GVL.TempSensError AND NOT .GVL.HumidSensEmerg AND NOT .GVL.PressBoundsEemrg AND NOT HeatEmerg AND .GVL.Mode=4 THEN
	.GVL.Emergency := FALSE;
	.GVL.Mode := 0;
END_IF

END_PROGRAM

// Device/Application/Humidifier
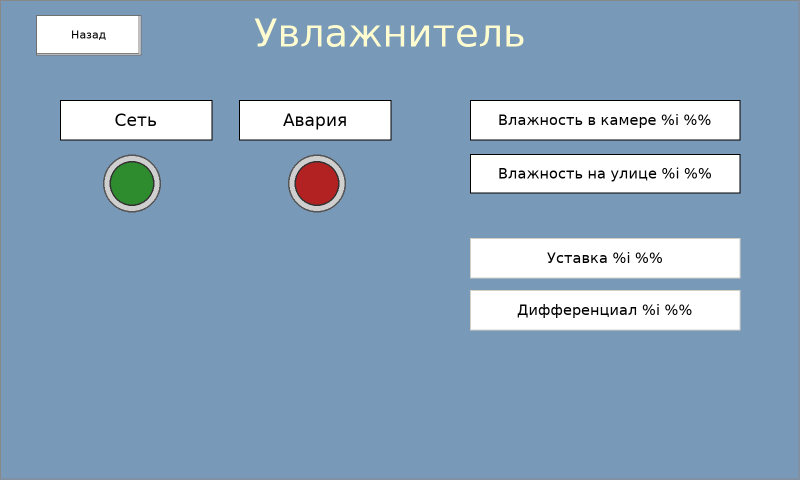
VISUALIZATION Humidifier  // 800x480
    Button (36,15 105x40), "Назад"
        OnMouseClick:  Assign=StartScreen, Type=Assignment
    Label (157,10 466x46), "Увлажнитель"
    Lamp1 (98,150 68x67), variable: GVL.InHumidPwr, style: Lamp-Lamp1-Green
    Lamp1 (283,150 68x67), variable: GVL.InHumidEmerg, style: Lamp-Lamp1-Red
    Rectangle (60,100 152x40), "Сеть"
    Rectangle (239,100 152x40), "Авария"
    Rectangle (470,100 270x40), "Влажность в камере %i %%", text variable: GVL.InAHumInside
    Rectangle (470,154 270x39), "Влажность на улице %i %%", text variable: GVL.InAHumOutside
    Textfield (470,238 270x40), "Уставка %i %%", text variable: PaintMode.HumidTarget
        OnMouseClick: write the text variable via Default, min 0, max 100
    Textfield (470,290 270x40), "Дифференциал %i %%", text variable: PaintMode.HumidDiff
        OnMouseClick: write the text variable via Default, min 0, max 100
END_VISUALIZATION

// Device/Application/Chiller
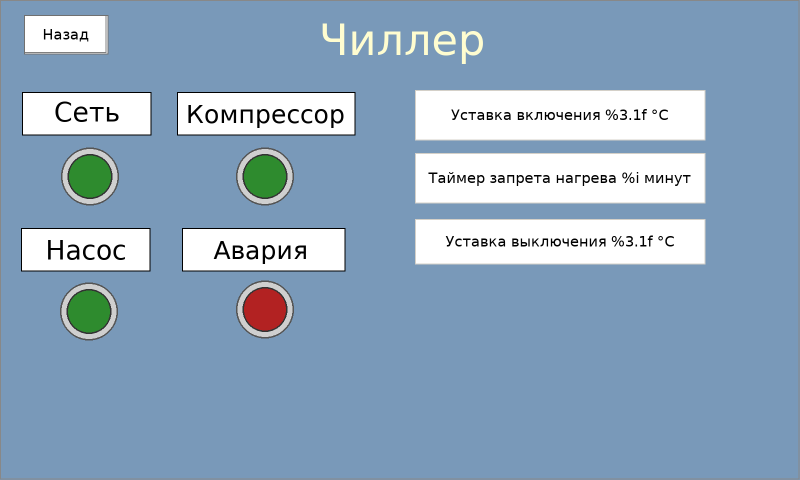
VISUALIZATION Chiller  // 800x480
    Lamp1 (56,143 68x67), variable: GVL.InChillerPwr, style: Lamp-Lamp1-Green
    Rectangle (22,92 129x43)
    Label (29,95 116x34), "Сеть"
    Lamp1 (55,278 68x67), variable: GVL.InChillerPump, style: Lamp-Lamp1-Green
    Rectangle (21,228 129x43)
    Label (28,233 116x34), "Насос"
    Lamp1 (231,143 68x67), variable: GVL.InChillerCompressor, style: Lamp-Lamp1-Green
    Rectangle (177,92 178x43)
    Label (181,97 169x34), "Компрессор"
    Lamp1 (231,276 68x67), variable: GVL.InChillerEmer, style: Lamp-Lamp1-Red
    Rectangle (182,228 163x43)
    Label (196,233 130x34), "Авария"
    Button (24,15 84x39), "Назад"
        OnMouseClick:  Assign=StartScreen, Type=Assignment
    Label (294,14 217x52), "Чиллер"
    Textfield (415,90 290x50), "Уставка включения %3.1f °C", text variable: PaintMode.ChillHDiff
        OnMouseClick: write the text variable via Default, min -50, max 150
    Textfield (415,219 290x45), "Уставка выключения %3.1f °C", text variable: PaintMode.ChillLDiff
        OnMouseClick: write the text variable via Default, min -50, max 150
    Textfield (415,153 290x50), "Таймер запрета нагрева %i минут", text variable: PaintMode.ChillCD
        OnMouseClick: write the text variable via Default, min -50, max 150
END_VISUALIZATION

// Device/Application/StartScreen
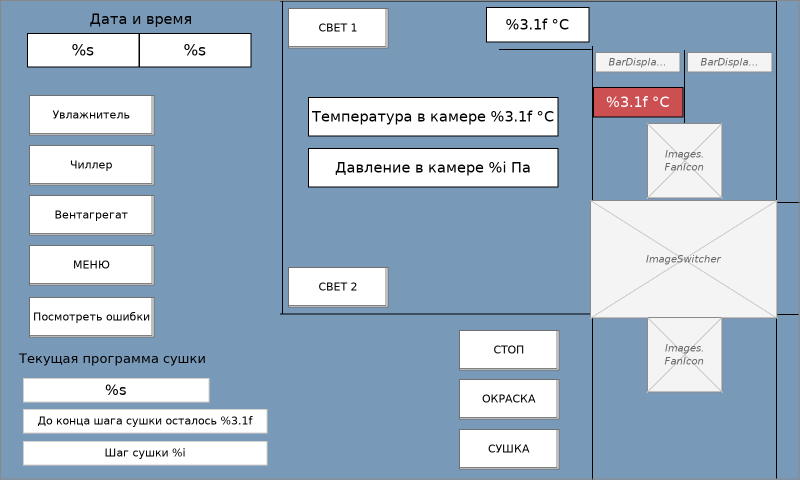
VISUALIZATION StartScreen  // 800x480
    Rectangle (593,87 90x30), "%3.1f °С", text variable: GVL.HExchangerFinalTemp
    Button (459,330 100x40), "СТОП"
        OnMouseClick: execute { .GVL.Mode := 0; }
    Button (459,379 100x40), "ОКРАСКА", colour toggle: PaintMode.PaintModeM
        p2175578022: PLC_PRG.dwOffColorToggle
        p573394764: PLC_PRG.ColorGreen
        OnMouseClick: execute {
            IF (.GVL.Mode = 0) THEN
            .GVL.Mode := 1;
            END_IF;
        }
    Button (459,429 100x40), "СУШКА", colour toggle: DryMode.DryModeM
        p2175578022: PLC_PRG.dwOffColorToggle
        p573394764: PLC_PRG.ColorGreen
        OnMouseClick: execute {
            IF (.GVL.Mode = 0) THEN
            	.GVL.Mode :=2;
            END_IF
        }
    Button (288,8 100x40), "СВЕТ 1", colour toggle: GVL.OutLight1
        p573394764: PLC_PRG.dwLightColorToggle
        p2175578022: PLC_PRG.dwOffColorToggle
        toggle GVL.OutLight1
    Button (288,267 100x40), "СВЕТ 2", colour toggle: GVL.OutLight2
        p573394764: PLC_PRG.dwLightColorToggle
        p2175578022: PLC_PRG.dwOffColorToggle
        toggle GVL.OutLight2
    Button (29,95 125x40), "Увлажнитель"
        p2175578022: Utils.CurrentHumidColor
        OnMouseClick:  Assign=Humidifier, Type=Assignment
    Button (29,145 125x40), "Чиллер"
        p2175578022: Utils.CurrentChillerColor
        OnMouseClick:  Assign=Chiller, Type=Assignment
    Button (29,195 125x40), "Вентагрегат"
        p2175578022: Utils.CurrentVentColor
        OnMouseClick:  Assign=VENT, Type=Assignment
    Button (29,245 125x40), "МЕНЮ"
        OnMouseClick:  Assign=MainMenu, Type=Assignment
    Rectangle (308,97 250x39), "Температура в камере %3.1f °C", text variable: GVL.ChamberFinalTemp
    Rectangle (308,148 250x39), "Давление в камере %i Па", text variable: GVL.InAChambPressure
    Rectangle (139,33 112x34), "%s", text variable: PLC_PRG.PLC_TIME
    Rectangle (27,33 112x34), "%s", text variable: PLC_PRG.PLC_DATE
    Label (43,1 196x36), "Дата и время"
    Label (23,346 179x25), "Текущая программа сушки"
    Textfield (23,378 186x24), "%s", text variable: DryMode.CurrentName
    Textfield (23,409 244x24), "До конца шага сушки осталось %3.1f", text variable: DryMode.StepTimeLeft
    Button (29,297 125x40), "Посмотреть ошибки"
        OnMouseClick:  Assign=Emergencies, Type=Assignment
    Textfield (23,441 244x24), "Шаг сушки %i", text variable: DryMode.index
    Line (800,431)
    Line (774,314) (799,314)
    Line (776,314) (776,479)
    Line (592,314) (592,480)
    Line (774,202) (800,202)
    Line (592,314) (280,314)
    Line (776,1) (280,1)
    Line (776,1) (776,202)
    Line (282,1) (282,314)
    Line (592,46) (592,200)
    Line (499,49) (591,49)
    Line (684,50) (684,125)
    ImageSwitcher (590,200 187x118), variable: Utils.ModeGateImg, input disabled if: Utils.DrivesOn, background image: Images.PaintIcon, image: Images.DryIcon, behaviour: TOGGLE
    Image (647,123 75x75), invisible if: Utils.NotInflowFan, image: Images.FanIcon
    Image (647,317 75x75), invisible if: Utils.NotExhaustFan, image: Images.FanIcon
    BarDisplayImage (595,52 85x20), value: GVL.inAFBCoolGate, style: BarDisplayImage-Gray, scale format: %.1f, scale 0..100
    BarDisplayImage (687,52 85x20), value: GVL.InAFBHeatGate, style: BarDisplayImage-Gray, scale format: %.1f, scale 0..100
    Rectangle (486,7 103x35), "%3.1f °С", text variable: GVL.EntryFinalTemp
END_VISUALIZATION

// Device/Application/MainMenu
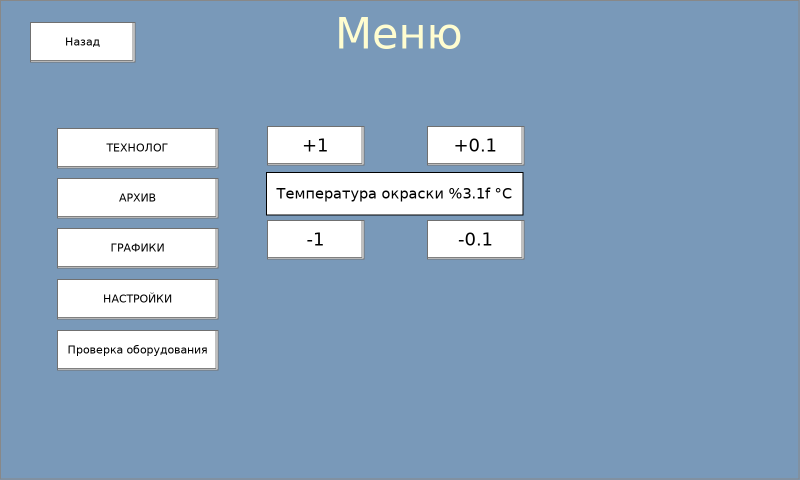
VISUALIZATION MainMenu  // 800x480
    Label (282,3 234x61), "Меню"
    Button (57,128 161x40), "ТЕХНОЛОГ"
        OnMouseClick:  Assign=DryProgs, Type=Assignment
    Button (57,178 161x40), "АРХИВ"
        OnMouseClick:  Assign=Archive, Type=Assignment
    Button (57,228 161x40), "ГРАФИКИ"
        OnMouseClick:  Assign=Trend, Type=Assignment
    Button (57,279 161x40), "НАСТРОЙКИ", image: Images.GearIcon
        OnMouseClick:  Assign=Settings, Type=Assignment
    Rectangle (266,172 257x43), "Температура окраски %3.1f °С", text variable: PaintMode.PaintPIDTarget
    Button (267,126 97x39), "+1"
        tap PaintMode.TempInc
    Button (267,220 97x39), "-1"
        tap PaintMode.TempDec
    Button (30,22 105x40), "Назад"
        OnMouseClick:  Assign=StartScreen, Type=Assignment
    Button (57,330 161x40), "Проверка оборудования"
        OnMouseClick:  Assign=DeviceCheck, Type=Assignment
    Button (427,126 97x39), "+0.1"
        tap PaintMode.TempIncS
    Button (427,220 97x39), "-0.1"
        tap PaintMode.TempDecS
END_VISUALIZATION

// Device/Application/Trend
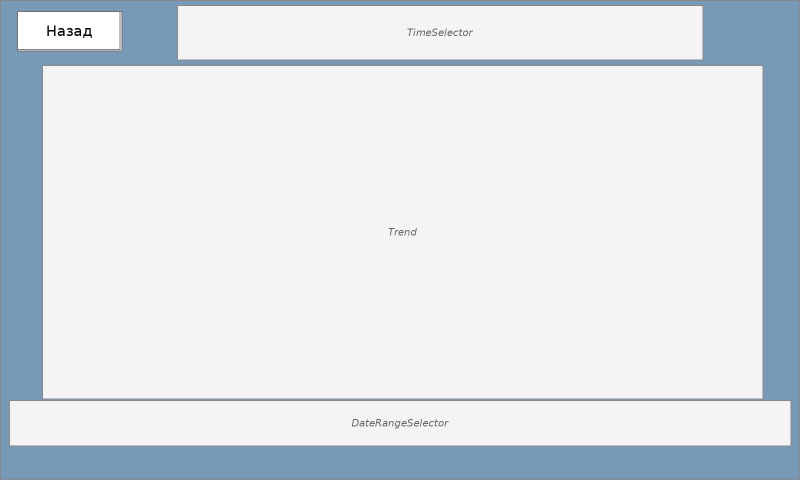
VISUALIZATION Trend  // 800x480
    Button (17,11 105x40), "Назад"
        OnMouseClick:  Assign=MainMenu, Type=Assignment
    Trend (42,65 721x334)
        p758368661: dd.MM.yyyy
        p2423372160: H:mm:ss:ms
        p2833066001: Trend_Trend1
        p2059293862: Trend1DateRangeSelector
        p2541140726: Trend1TimeSelector
    DateRangeSelector (9,400 782x46)
        p1661464551: GenElemInst_8
    TimeSelector (177,5 526x55)
        p3737533738: GenElemInst_8
        p677259794: Zoom:
END_VISUALIZATION

// Device/Application/VENT
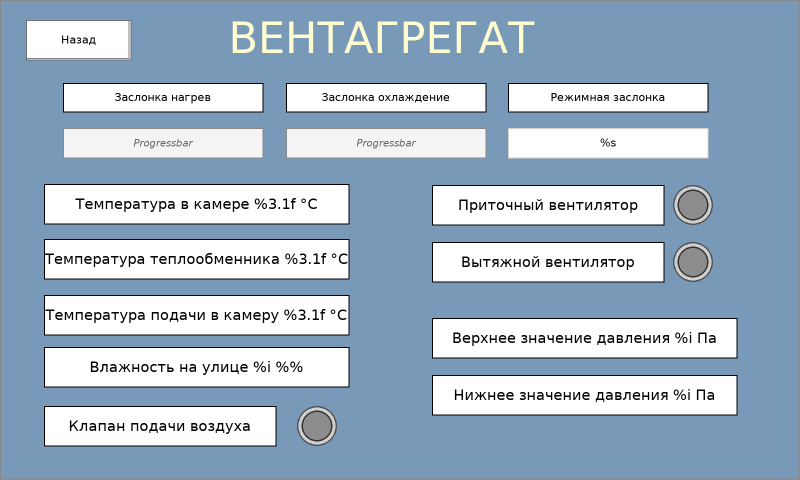
VISUALIZATION VENT  // 800x480
    Label (209,12 345x52), "ВЕНТАГРЕГАТ"
    Button (26,20 105x40), "Назад"
        OnMouseClick:  Assign=StartScreen, Type=Assignment
    Progressbar (63,128 200x30), variable: GVL.InAFBHeatGate
    Rectangle (63,83 200x29), "Заслонка нагрев"
    Progressbar (286,128 200x30), variable: GVL.inAFBCoolGate
    Rectangle (286,83 200x29), "Заслонка охлаждение"
    Textfield (508,128 200x30), "%s", text variable: Utils.GateMode
    Rectangle (508,83 200x29), "Режимная заслонка"
    Rectangle (44,184 305x40), "Температура в камере %3.1f °С", text variable: GVL.ChamberFinalTemp
    Rectangle (44,239 305x40), "Температура теплообменника %3.1f °С", text variable: GVL.HExchangerFinalTemp
    Rectangle (44,347 305x40), "Влажность на улице %i %%", text variable: GVL.InAHumOutside
    Rectangle (44,295 305x40), "Температура подачи в камеру %3.1f °С", text variable: GVL.EntryFinalTemp
    Rectangle (44,406 232x40), "Клапан подачи воздуха"
    Lamp1 (294,403 46x46), variable: GVL.OutAirPump, style: Lamp-Lamp1-Gray
    Rectangle (432,185 232x40), "Приточный вентилятор"
    Lamp1 (670,182 46x46), variable: GVL.OutInflowFan, style: Lamp-Lamp1-Gray
    Rectangle (432,242 232x40), "Вытяжной вентилятор"
    Lamp1 (670,239 46x46), variable: GVL.OutExhaustFan, style: Lamp-Lamp1-Gray
    Rectangle (432,318 305x40), "Верхнее значение давления %i Па", text variable: Utils.PressureHigh
        OnMouseClick: write the text variable via Default, min 0, max 250
    Rectangle (432,375 305x40), "Нижнее значение давления %i Па", text variable: Utils.PressureLow
        OnMouseClick: write the text variable via Default, min 0, max 250
END_VISUALIZATION

// Device/Application/Settings
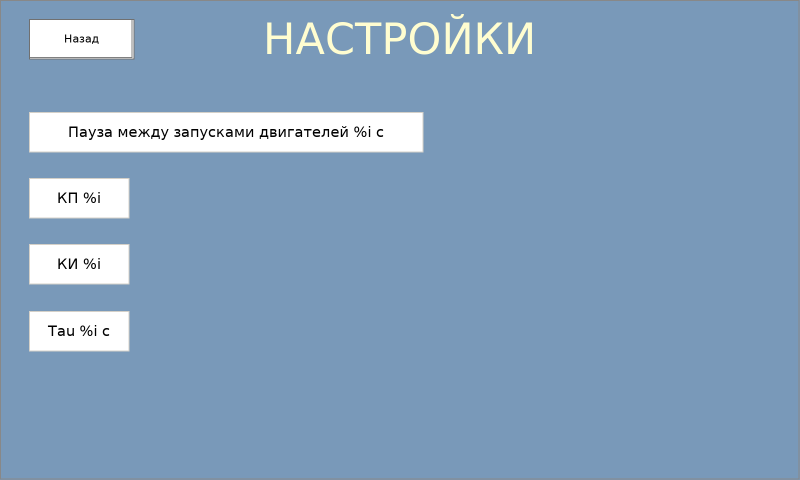
VISUALIZATION Settings  // 800x480
    Label (227,13 345x52), "НАСТРОЙКИ"
    Textfield (29,112 394x40), "Пауза между запусками двигателей %i с", text variable: GVL.ExhFanD
        OnMouseClick: write the text variable via Default, min 0, max 100
    Textfield (29,178 100x40), "КП %i", text variable: PID_controller.KP
        OnMouseClick: write the text variable via Default, min 0, max 100
    Textfield (29,244 100x40), "КИ %i", text variable: PID_controller.KI
        OnMouseClick: write the text variable via Default, min 0, max 100
    Textfield (29,311 100x40), "Tau %i c", text variable: PID_controller.Tau
        OnMouseClick: write the text variable via Default, min 0, max 100
    Button (29,19 105x40), "Назад"
        OnMouseClick:  Assign=MainMenu, Type=Assignment
END_VISUALIZATION

// Device/Application/DryProgs
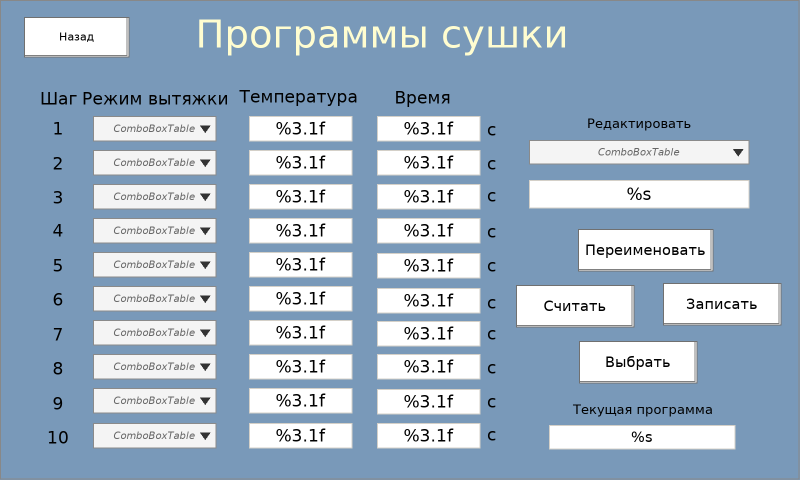
VISUALIZATION DryProgs  // 800x480
    Label (83,86 145x25), "Режим вытяжки"
    Label (230,84 138x25), "Температура"
    Label (358,85 129x25), "Время"
    Label (34,86 50x25), "Шаг"
    Label (33,116 50x25), "1"
    Label (33,151 50x25), "2"
    Label (33,185 50x25), "3"
    Label (33,218 50x25), "4"
    Label (33,253 50x25), "5"
    Label (33,287 50x25), "6"
    Label (33,322 50x25), "7"
    Label (33,356 50x25), "8"
    Label (33,391 50x25), "9"
    Label (33,425 50x25), "10"
    ComboBoxTable (93,116 123x25), variable: DryMode.Buffer[1,1], data array: DryMode.Modes
        p3854506369: DryMode.Modes[INDEX]
    ComboBoxTable (93,150 123x25), variable: DryMode.Buffer[1,2], data array: DryMode.Modes
        p3854506369: DryMode.Modes[INDEX]
    ComboBoxTable (93,184 123x25), variable: DryMode.Buffer[1,3], data array: DryMode.Modes
        p3854506369: DryMode.Modes[INDEX]
    ComboBoxTable (93,218 123x25), variable: DryMode.Buffer[1,4], data array: DryMode.Modes
        p3854506369: DryMode.Modes[INDEX]
    ComboBoxTable (93,252 123x25), variable: DryMode.Buffer[1,5], data array: DryMode.Modes
        p3854506369: DryMode.Modes[INDEX]
    ComboBoxTable (93,286 123x25), variable: DryMode.Buffer[1,6], data array: DryMode.Modes
        p3854506369: DryMode.Modes[INDEX]
    ComboBoxTable (93,320 123x25), variable: DryMode.Buffer[1,7], data array: DryMode.Modes
        p3854506369: DryMode.Modes[INDEX]
    ComboBoxTable (93,354 123x25), variable: DryMode.Buffer[1,8], data array: DryMode.Modes
        p3854506369: DryMode.Modes[INDEX]
    ComboBoxTable (93,388 123x25), variable: DryMode.Buffer[1,9], data array: DryMode.Modes
        p3854506369: DryMode.Modes[INDEX]
    ComboBoxTable (93,423 123x25), variable: DryMode.Buffer[1,10], data array: DryMode.Modes
        p3854506369: DryMode.Modes[INDEX]
    Textfield (377,423 103x25), "%3.1f", text variable: DryMode.Buffer[3,10]
        OnMouseClick: write the text variable via Default, min 0, max 100
    Textfield (249,423 103x25), "%3.1f", text variable: DryMode.Buffer[2,10]
        OnMouseClick: write the text variable via Default, min -50, max 200
    Textfield (377,116 103x25), "%3.1f", text variable: DryMode.Buffer[3,1]
        OnMouseClick: write the text variable via Default, min 0, max 100
    Textfield (249,116 103x25), "%3.1f", text variable: DryMode.Buffer[2,1]
        OnMouseClick: write the text variable via Default, min -50, max 200
    Textfield (377,150 103x25), "%3.1f", text variable: DryMode.Buffer[3,2]
        OnMouseClick: write the text variable via Default, min 0, max 100
    Textfield (249,150 103x25), "%3.1f", text variable: DryMode.Buffer[2,2]
        OnMouseClick: write the text variable via Default, min -50, max 200
    Textfield (377,184 103x25), "%3.1f", text variable: DryMode.Buffer[3,3]
        OnMouseClick: write the text variable via Default, min 0, max 100
    Textfield (249,184 103x25), "%3.1f", text variable: DryMode.Buffer[2,3]
        OnMouseClick: write the text variable via Default, min -50, max 200
    Textfield (377,218 103x25), "%3.1f", text variable: DryMode.Buffer[3,4]
        OnMouseClick: write the text variable via Default, min 0, max 100
    Textfield (249,218 103x25), "%3.1f", text variable: DryMode.Buffer[2,4]
        OnMouseClick: write the text variable via Default, min -50, max 200
    Textfield (377,253 103x25), "%3.1f", text variable: DryMode.Buffer[3,5]
        OnMouseClick: write the text variable via Default, min 0, max 100
    Textfield (249,252 103x25), "%3.1f", text variable: DryMode.Buffer[2,5]
        OnMouseClick: write the text variable via Default, min -50, max 200
    Textfield (377,288 103x25), "%3.1f", text variable: DryMode.Buffer[3,6]
        OnMouseClick: write the text variable via Default, min 0, max 100
    Textfield (249,286 103x25), "%3.1f", text variable: DryMode.Buffer[2,6]
        OnMouseClick: write the text variable via Default, min -50, max 200
    Textfield (377,321 103x25), "%3.1f", text variable: DryMode.Buffer[3,7]
        OnMouseClick: write the text variable via Default, min 0, max 100
    Textfield (249,320 103x25), "%3.1f", text variable: DryMode.Buffer[2,7]
        OnMouseClick: write the text variable via Default, min -50, max 200
    Textfield (377,354 103x25), "%3.1f", text variable: DryMode.Buffer[3,8]
        OnMouseClick: write the text variable via Default, min 0, max 100
    Textfield (249,354 103x25), "%3.1f", text variable: DryMode.Buffer[2,8]
        OnMouseClick: write the text variable via Default, min -50, max 200
    Textfield (377,389 103x25), "%3.1f", text variable: DryMode.Buffer[3,9]
        OnMouseClick: write the text variable via Default, min 0, max 100
    Textfield (249,388 103x25), "%3.1f", text variable: DryMode.Buffer[2,9]
        OnMouseClick: write the text variable via Default, min -50, max 200
    Button (24,17 105x40), "Назад"
        OnMouseClick:  Assign=MainMenu, Type=Assignment
    Label (149,11 466x46), "Программы сушки"
    Label (467,117 50x25), "c"
    Label (467,151 50x25), "c"
    Label (467,183 50x25), "c"
    Label (467,219 50x25), "c"
    Label (467,253 50x25), "c"
    Label (467,290 50x25), "c"
    Label (467,321 50x25), "c"
    Label (467,355 50x25), "c"
    Label (467,389 50x25), "c"
    Label (467,422 50x25), "c"
    ComboBoxTable (529,140 220x24), variable: DryMode.SelectedProg, data array: DryMode.Progs
        p3854506369: DryMode.Progs[INDEX]
    Button (516,285 118x42), "Считать"
        tap DryMode.ProgChanged
    Label (570,111 138x25), "Редактировать"
    Textfield (529,180 220x28), "%s", text variable: DryMode.NewName
        OnMouseClick: write the text variable via VisuKbEnRu.Keypad
    Button (663,283 118x42), "Записать"
        tap DryMode.ProgSave
    Button (578,229 135x42), "Переименовать"
        tap DryMode.SaveName
    Button (579,341 118x42), "Выбрать"
        tap DryMode.ChooseProg
    Label (567,397 152x25), "Текущая программа"
    Textfield (549,425 186x24), "%s", text variable: DryMode.CurrentName
END_VISUALIZATION

// Device/Application/DeviceCheck
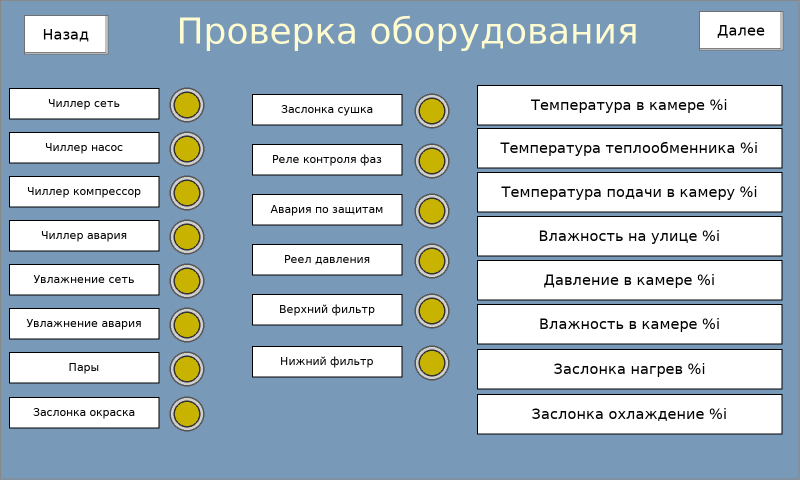
VISUALIZATION DeviceCheck  // 800x480
    Button (24,15 84x39), "Назад"
        OnMouseClick:  Assign=MainMenu, Type=Assignment
    Label (173,5 469x52), "Проверка оборудования"
    Lamp1 (167,85 40x40), variable: GVL.InChillerPwr, style: Lamp-Lamp1-Yellow
    Rectangle (477,85 305x40), "Температура в камере %i", text variable: GVL.InAChamberTemp
    Rectangle (477,128 305x40), "Температура теплообменника %i", text variable: GVL.InAHExchanger
    Rectangle (477,216 305x40), "Влажность на улице %i", text variable: GVL.InAHumOutside
    Rectangle (477,172 305x40), "Температура подачи в камеру %i", text variable: GVL.InAEntryTemp
    Rectangle (477,260 305x40), "Давление в камере %i", text variable: GVL.InAChambPressure
    Rectangle (477,304 305x40), "Влажность в камере %i", text variable: GVL.InAHumInside
    Rectangle (477,394 305x40), "Заслонка охлаждение %i", text variable: GVL.inAFBCoolGate
    Rectangle (477,349 305x40), "Заслонка нагрев %i", text variable: GVL.InAFBHeatGate
    Rectangle (9,88 150x31), "Чиллер сеть"
    Lamp1 (167,129 40x40), variable: GVL.InChillerPump, style: Lamp-Lamp1-Yellow
    Rectangle (9,132 150x31), "Чиллер насос"
    Lamp1 (167,173 40x40), variable: GVL.InChillerCompressor, style: Lamp-Lamp1-Yellow
    Rectangle (9,176 150x31), "Чиллер компрессор"
    Lamp1 (167,261 40x40), variable: GVL.InHumidPwr, style: Lamp-Lamp1-Yellow
    Rectangle (9,264 150x31), "Увлажнение сеть"
    Lamp1 (167,305 40x40), variable: GVL.InHumidEmerg, style: Lamp-Lamp1-Yellow
    Rectangle (9,308 150x31), "Увлажнение авария"
    Lamp1 (167,349 40x40), variable: GVL.InFireSteam, style: Lamp-Lamp1-Yellow
    Rectangle (9,352 150x31), "Пары"
    Lamp1 (167,394 40x40), variable: GVL.InModeGatePaint, style: Lamp-Lamp1-Yellow
    Rectangle (9,397 150x31), "Заслонка окраска"
    Lamp1 (412,91 40x40), variable: GVL.InModeGateDry, style: Lamp-Lamp1-Yellow
    Rectangle (252,94 150x31), "Заслонка сушка"
    Lamp1 (412,141 40x40), variable: GVL.InPhaseControl, style: Lamp-Lamp1-Yellow
    Rectangle (252,144 150x31), "Реле контроля фаз"
    Lamp1 (412,191 40x40), variable: GVL.InNetEmerg, style: Lamp-Lamp1-Yellow
    Rectangle (252,194 150x31), "Авария по защитам"
    Lamp1 (412,241 40x40), variable: GVL.InChamberPressure, style: Lamp-Lamp1-Yellow
    Rectangle (252,244 150x31), "Реел давления"
    Lamp1 (412,291 40x40), variable: GVL.InUpperFilter, style: Lamp-Lamp1-Yellow
    Rectangle (252,294 150x31), "Верхний фильтр"
    Lamp1 (412,343 40x40), variable: GVL.InLowerFilter, style: Lamp-Lamp1-Yellow
    Rectangle (252,346 150x31), "Нижний фильтр"
    Lamp1 (167,217 40x40), variable: GVL.InChillerEmer, style: Lamp-Lamp1-Yellow
    Rectangle (9,220 150x31), "Чиллер авария"
    Button (699,11 84x39), "Далее", invisible if: Utils.ManualBlock
        OnMouseClick:  Assign=DeviceCheck_2, Type=Assignment
END_VISUALIZATION

// Device/Application/DeviceCheck_2
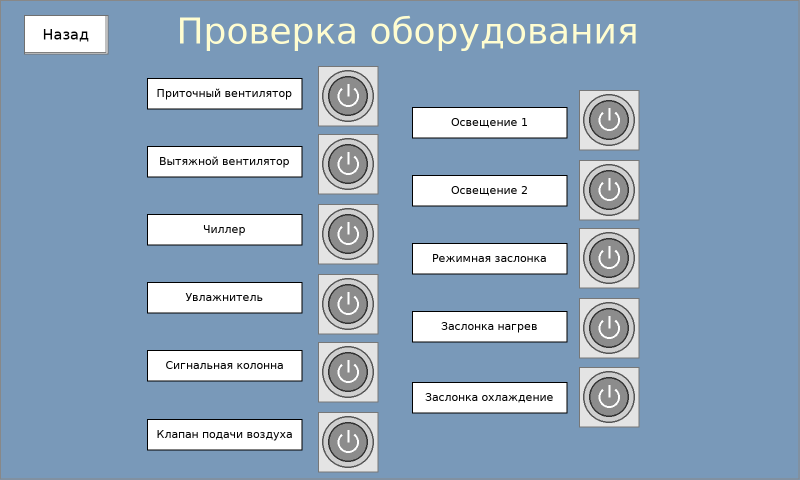
VISUALIZATION DeviceCheck_2  // 800x480
    Button (24,15 84x39), "Назад"
        OnMouseClick:  Assign=DeviceCheck, Type=Assignment
    Label (173,5 469x52), "Проверка оборудования"
    PowerSwitch (318,66 60x60), variable: GVL.OutInflowFan, behaviour: TOGGLE, style: Switch-PowerSwitch-Gray
    Rectangle (147,78 155x31), "Приточный вентилятор"
    Rectangle (147,146 155x31), "Вытяжной вентилятор"
    Rectangle (147,214 155x31), "Чиллер"
    Rectangle (147,282 155x31), "Увлажнитель"
    Rectangle (147,350 155x31), "Сигнальная колонна"
    Rectangle (412,107 155x31), "Освещение 1"
    Rectangle (412,175 155x31), "Освещение 2"
    Rectangle (412,243 155x31), "Режимная заслонка"
    Rectangle (412,311 155x31), "Заслонка нагрев"
    Rectangle (147,419 155x31), "Клапан подачи воздуха"
    Rectangle (412,382 155x31), "Заслонка охлаждение"
    PowerSwitch (318,134 60x60), variable: GVL.OutExhaustFan, behaviour: TOGGLE, style: Switch-PowerSwitch-Gray
    PowerSwitch (318,204 60x60), variable: GVL.OutChiller, behaviour: TOGGLE, style: Switch-PowerSwitch-Gray
    PowerSwitch (318,274 60x60), variable: GVL.OutHumid, behaviour: TOGGLE, style: Switch-PowerSwitch-Gray
    PowerSwitch (318,342 60x60), variable: GVL.OutEmergLamp, behaviour: TOGGLE, style: Switch-PowerSwitch-Gray
    PowerSwitch (318,412 60x60), variable: GVL.OutAirPump, behaviour: TOGGLE, style: Switch-PowerSwitch-Gray
    PowerSwitch (579,90 60x60), variable: GVL.OutLight1, behaviour: TOGGLE, style: Switch-PowerSwitch-Gray
    PowerSwitch (579,160 60x60), variable: GVL.OutLight2, behaviour: TOGGLE, style: Switch-PowerSwitch-Gray
    PowerSwitch (579,228 60x60), variable: GVL.OutModeGate, behaviour: TOGGLE, style: Switch-PowerSwitch-Gray
    PowerSwitch (579,298 60x60), variable: GVL.OutHeatGate, behaviour: TOGGLE, style: Switch-PowerSwitch-Gray
    PowerSwitch (579,367 60x60), variable: GVL.OutCoolGate, behaviour: TOGGLE, style: Switch-PowerSwitch-Gray
END_VISUALIZATION

// Device/Application/Archive
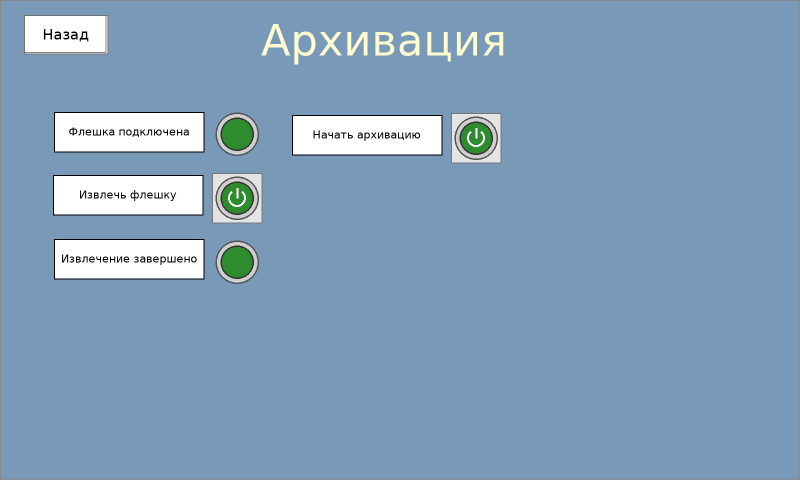
VISUALIZATION Archive  // 800x480
    Button (24,15 84x39), "Назад"
        OnMouseClick:  Assign=MainMenu, Type=Assignment
    Label (233,8 302x65), "Архивация"
    Rectangle (54,112 150x40), "Флешка подключена"
    Lamp1 (212,109 50x50), variable: PLC_PRG.USBMounted, style: Lamp-Lamp1-Green
    PowerSwitch (212,173 50x50), variable: PLC_PRG.USBUnmount, behaviour: TOGGLE, style: Switch-PowerSwitch-Green
    Rectangle (53,175 150x40), "Извлечь флешку"
    Rectangle (54,239 150x40), "Извлечение завершено"
    Lamp1 (212,237 50x50), variable: PLC_PRG.USBUnmountDone, style: Lamp-Lamp1-Green
    PowerSwitch (451,113 50x50), variable: PLC_PRG.StartArchive, behaviour: TOGGLE, style: Switch-PowerSwitch-Green
    Rectangle (292,115 150x40), "Начать архивацию"
END_VISUALIZATION

// Device/Application/Emergencies
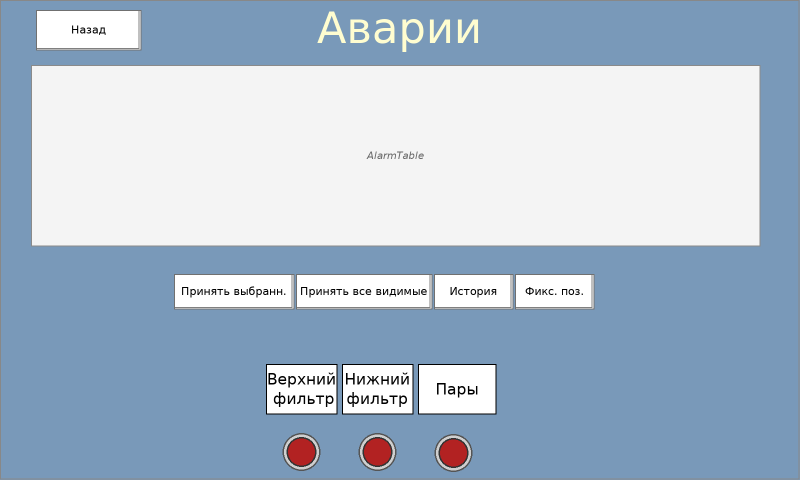
VISUALIZATION Emergencies  // 800x480
    Lamp1 (279,430 45x44), variable: Emrg.UpperFilterOut, style: Lamp-Lamp1-Red
    Lamp1 (355,430 45x44), variable: Emrg.LowerFilterOut, style: Lamp-Lamp1-Red
    AlarmTable (31,65 729x181)
        p1521930926: __All
        p1663851261: __All
        p428520879: Emrg.AcknSelected
        p2607059081: Emrg.AcknVisible
        p3266827225: Emrg.EmergHistory
        p3894972949: Emrg.EmergFixedPos
    Lamp1 (431,431 45x44), variable: GVL.InFireSteam, style: Lamp-Lamp1-Red
    Rectangle (418,364 78x50), "Пары", text variable: PLC_PRG.PLC_DATE
    Rectangle (266,364 71x50), "Верхний фильтр", text variable: PLC_PRG.PLC_DATE
    Rectangle (342,364 71x50), "Нижний фильтр", text variable: PLC_PRG.PLC_DATE
    Button (174,274 120x35), "Принять выбранн."
        toggle Emrg.AcknSelected
    Button (296,274 136x35), "Принять все видимые"
        toggle Emrg.AcknVisible
    Button (434,274 79x35), "История"
        toggle Emrg.EmergHistory
    Button (515,274 79x35), "Фикс. поз."
        toggle Emrg.EmergFixedPos
    Button (36,10 105x40), "Назад"
        OnMouseClick:  Assign=StartScreen, Type=Assignment
    Label (250,3 299x50), "Аварии"
END_VISUALIZATION

(* text list Emergencies (id | default)
  6 | Ошибка давления в камере
  5 | Ошибка датчика влажности
  4 | Ошибка датчика температуры
  3 | Реле давления
  2 | Нет нагрева
  1 | Аваря по реле контроля фаз
  0 | Авария по защитам
   |  *)
